// TIA Portal V17 export
// export: Created 2025-03-10T12:14:34.5546891Z, ExportSetting WithDefaults, DisplayName Totally Integrated Automation Portal, DisplayVersion V17 Update 8, DisplayName TIA Portal Openness, DisplayVersion V17 Update 8, DisplayName TIA Portal Version Control Interface, DisplayVersion V17, DisplayName SINAMICS Startdrive Advanced, DisplayVersion V17 SP2, DisplayName SINAMICS Startdrive G110M, G120, G120C, G120D, G120P, G115D, DisplayVersion V17 SP2, DisplayName SINAMICS Startdrive G130, G150, S120, S150, SINAMICS MV, S210, DisplayVersion V17 SP2, DisplayName STEP 7 Professional, DisplayVersion V17 Update 8, DisplayName SINUMERIK ONE STEP 7 Toolbox, DisplayVersion V17 Update 12, DisplayName SINUMERIK 840D sl STEP 7 Toolbox, DisplayVersion V17 Update 12, DisplayName STEP 7 Safety, DisplayVersion V17 Update 6, DisplayName WinCC Advanced, DisplayVersion V17 Update 8
DATA_BLOCK "LBP_ConfigData"   // DB7
TITLE = Configuration parameter / Parámetros de configuración / Konfigurationsparameter
{ S7_Optimized_Access := 'FALSE'; DB_Accessible_From_OPC_UA := 'FALSE' }
AUTHOR : SINUMERIK
FAMILY : SINUMERIK_ONE
VERSION : 6.15
// Contains parameters for the configuration and initialization of the basic program / Contiene parámetros para la configuración e inicialización del programa básico / Enthält Parameter für die Konfiguration und Initialisierung des Grundprogramms
// stored: AutoNumber false, DBAccessibleFromOPCUA false, DBAccessibleFromWebserver true, InstanceOfName LBP_typeConfigData, InstanceOfType UDT, IsOnlyStoredInLoadMemory false, IsWriteProtectedInAS false
"LBP_typeConfigData"
   // VAR RETAIN
   //    MCPNum : Int;
   //    MCP1In : Struct
   //       DBNo : Word;
   //       Addr : DWord;
   //    END_STRUCT;
   //    MCP1Out : Struct
   //       DBNo : Word;
   //       Addr : DWord;
   //    END_STRUCT;
   //    reservedByte14_25 : Array[14..25] of Byte;
   //    MCP1BusAdr : Int;
   //    MCP1Timeout : S5Time;
   //    reservedByte30_31 : Array[30..31] of Byte;
   //    MCP2In : Struct
   //       DBNo : Word;
   //       Addr : DWord;
   //    END_STRUCT;
   //    MCP2Out : Struct
   //       DBNo : Word;
   //       Addr : DWord;
   //    END_STRUCT;
   //    reservedByte44_55 : Array[44..55] of Byte;
   //    MCP2BusAdr : Int;
   //    MCP2Timeout : S5Time;
   //    reservedByte60_61 : Array[60..61] of Byte;
   //    reservedBool62_0 : Bool;
   //    MCP1Stop : Bool;
   //    MCP2Stop : Bool;
   //    MCP1NotSend : Bool;
   //    MCP2NotSend : Bool;
   //    reservedBool62_5 : Bool;
   //    reservedBool62_6 : Bool;
   //    MCPBusType : Byte;
   //    HTIf : Int;
   //    HTIn : Struct
   //       DBNo : Word;
   //       Addr : DWord;
   //    END_STRUCT;
   //    HTOut : Struct
   //       DBNo : Word;
   //       Addr : DWord;
   //    END_STRUCT;
   //    reservedByte78_95 : Array[78..95] of Byte;
   //    HTAdr : Int;
   //    reservedByte98_107 : Array[98..107] of Byte;
   //    reservedBool108_0 : Bool;
   //    HTStop : Bool;
   //    HTNotSend : Bool;
   //    NCCyclTimeout : S5Time;
   //    NCRunupTimeout : S5Time;
   //    ListMDecGrp : Int;
   //    reservedBool116_0 : Bool;
   //    MMCToIF : Bool;
   //    HWheelMMC : Bool;
   //    reservedBool116_3 : Bool;
   //    MCP_IF_TCS : Bool;
   //    ExtendChanAxMsg : Bool;
   //    HMIAxisSel : Bool;
   //    DeactivateCtrlEnergy : Bool;
   //    MsgUser : Int;
   //    reservedBool120_0 : Bool;
   //    IRAuxfuT : Bool;
   //    IRAuxfuH : Bool;
   //    IRAuxfuE : Bool;
   //    UserVersion : Struct
   //       DBNo : Word;
   //       Addr : DWord;
   //    END_STRUCT;
   //    OpKeyNum : Int;
   //    Op1KeyIn : Struct
   //       DBNo : Word;
   //       Addr : DWord;
   //    END_STRUCT;
   //    Op1KeyOut : Struct
   //       DBNo : Word;
   //       Addr : DWord;
   //    END_STRUCT;
   //    Op1KeyBusAdr : Int;
   //    Op2KeyIn : Struct
   //       DBNo : Word;
   //       Addr : DWord;
   //    END_STRUCT;
   //    Op2KeyOut : Struct
   //       DBNo : Word;
   //       Addr : DWord;
   //    END_STRUCT;
   //    Op2KeyBusAdr : Int;
   //    Op1KeyStop : Bool;
   //    Op2KeyStop : Bool;
   //    Op1KeyNotSend : Bool;
   //    Op2KeyNotSend : Bool;
   //    reservedByte159 : Byte;
   //    IdentMcpBusAdr : Int;
   //    IdentMcpProfilNo : Byte;
   //    IdentMcpBusType : Byte;
   //    IdentMcpStrobe : Bool;
   //    MaxModeGroup : Int;
   //    MaxChan : Int;
   //    MaxAxis : Int;
   //    ActiveChan : Array[1..10] of Bool;
   //    ActiveAxis : Array[1..31] of Bool;
   //    MaxNumUserDataInt : Int;
   //    MaxNumUserDataHex : Int;
   //    MaxNumUserDataReal : Int;
   //    IdentMcpType : Byte;
   //    IdentMcpLengthIn : Byte;
   //    IdentMcpLengthOut : Byte;
   //    reservedByte188_199 : Array[188..199] of Byte;
   //    LBPVersionInfo : String[44] := 'SINUMERIK ONE V06.15.00.03.001 18/01/23 $L';
   //    UserVersionInfo : String[44];
   //    GenerateAlarmMsgs : Struct
   //       NumActAlarmMsgs : UInt;
   //       Error : Bool;
   //       StatusID : UInt;
   //       Status : Word;
   //    END_STRUCT;
   //    OpUnitCommId : UInt;
   //    OpUnitInterfaceId : HW_ANY;
   //    MCP1ConnectionId : CONN_OUC;
   //    MCP2ConnectionId : CONN_OUC;
   //    HTConnectionId : CONN_OUC;
   //    Op1KeyConnectionId : CONN_OUC;
   //    Op2KeyConnectionId : CONN_OUC;
   //    IdentConnectionId : CONN_OUC;
   //    MCP1LocalUdpPort : UInt;
   //    MCP2LocalUdpPort : UInt;
   //    HTLocalUdpPort : UInt;
   //    Op1KeyLocalUdpPort : UInt;
   //    Op2KeyLocalUdpPort : UInt;
   //    IdentLocalUdpPort : UInt;
   //    MCP1Error : Bool;
   //    MCP1Status : Word;
   //    MCP2Error : Bool;
   //    MCP2Status : Word;
   //    HTError : Bool;
   //    HTStatus : Word;
   //    Op1KeyError : Bool;
   //    Op1KeyStatus : Word;
   //    Op2KeyError : Bool;
   //    Op2KeyStatus : Word;
   //    IdentError : Bool;
   //    IdentStatus : Word;
   //    MCP1Ready : Bool;
   //    MCP2Ready : Bool;
   //    HTReady : Bool;
   //    Op1KeyReady : Bool;
   //    Op2KeyReady : Bool;
   // END_VAR
BEGIN
END_DATA_BLOCK
